{attribute 'qualified_only'}
// Owner-local, bounded publication of the demo's physical CX2030 I/O tree.
// ST_IoChannel.Name is always the exact electrical-list/schematic tag.
VAR_GLOBAL
    {attribute 'OPC.UA.DA' := '1'}
    Topology : ST_FieldbusTopology;
END_VAR

(* stored: Version 1.1.0.1, ProductVersion 3.1.4024.12
   GVL GVL_PressFieldbus: Id {a3646726-391b-4c93-950c-6c1282fdb93f} *)
